(* PLC project LadderExecuteFixture, greenforge-labs codescribe-fixture 1 *)
(* stored: creationDateTime 2020-01-01T00:00:00 *)

PROGRAM LD_EXECUTE
  VAR
    xSet : BOOL;
    xClear : BOOL;
    xCount : BOOL;
    xDone : BOOL;
  END_VAR

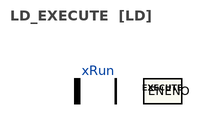
(* LD diagram, written out as Structured Text *)
IF xRun THEN
  iCount := iCount + 1;
  IF iCount > 10 THEN
  iCount := 0;
  END_IF
END_IF;
END_PROGRAM
